FUNCTION_BLOCK Q_EndPoint (* Command change end point ( Part 6 - F.26 ) *)
  (* Standard: ISO 11783-6; Description: This command is used to change the end point of a line object by changing the width, height and/or line direction attributes. Return values iso_s16 - E_NO_ERR - OK - E_OVERFLOW - buffer overflow - E_NOACT - Command not possible in current state - E_NO_INSTANCE - No VT client available *)
  (* Version 1.0, 2022-07-08, franz *)
  (* Documentation:
  This command is used to change the end point of a line object by changing the width, height and/or line direction attributes.
   Return values
   iso_s16
    - E_NO_ERR - OK
   - E_OVERFLOW - buffer overflow
   - E_NOACT - Command not possible in current state
   - E_NO_INSTANCE - No VT client available
  *)
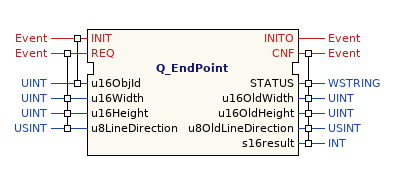
  EVENT_INPUT
    INIT WITH u16ObjId; (* Service Initialization *)
    REQ WITH u16Width, u16Height, u8LineDirection; (* Service Request *)
  END_EVENT
  EVENT_OUTPUT
    INITO; (* Initialization Confirm *)
    CNF WITH STATUS, u8OldLineDirection, u16OldWidth, u16OldHeight, s16result; (* Confirmation of Requested Service *)
  END_EVENT
  VAR_INPUT
    u16ObjId : UINT; (* Object ID *)
    u16Width : UINT; (* X value of end point *)
    u16Height : UINT; (* Y value of end point *)
    u8LineDirection : USINT; (* Line direction see Part 6 - B.27 *)
  END_VAR
  VAR_OUTPUT
    STATUS : WSTRING; (* Service Status *)
    u16OldWidth : UINT; (* Old X value of end point *)
    u16OldHeight : UINT; (* Old Y value of end point *)
    u8OldLineDirection : USINT; (* Old line direction see Part 6 - B.27 *)
    s16result : INT; (* retval see description *)
  END_VAR
END_FUNCTION_BLOCK
